// TIA Portal V20 export
DATA_BLOCK "DB_Manual"   // DB18
// stored: Access Published, MemoryReserve 100, Namespace LineB1
   VAR
      Conveyor : Struct
         ID : Int;
         Enable : Bool;
         Run : Bool;
         in : Bool;
      END_STRUCT;
      Line : Struct
         B1 : Struct
            Conveyor { S7_SetPoint := 'True'} : Array[_.minB1.._.maxB1] of "LineB1.ManualInputs";
         END_STRUCT;
      END_STRUCT;
   END_VAR
BEGIN
END_DATA_BLOCK
